TYPE T_ControllerValue : LREAL; END_TYPE

(* stored: Version 1.1.0.1, ProductVersion 3.1.4024.14
   DUT T_ControllerValue: Id {d62ed199-f9c3-0652-3311-e2ec5065d824} *)
